{attribute 'qualified_only'}
VAR_GLOBAL
	rMoisture : REAL :=50; // Represent the soil moisture
	rTemp : REAL := 25; // Shows the temperature in Celsius
	bWaterRequired : BOOL := FALSE; // Tells if water is needed
	bWaterON : BOOL := FALSE; // Pump is on
	tWaterTimer : TIME :=T#0s // Tell watering period
END_VAR

(* stored: Version 1.1.0.1, ProductVersion 3.1.4024.15
   GVL GVL: Id {43c0d85a-6909-422a-aaef-bb46a75b5c35} *)
